TYPE "ST_SpkUnitHal"
VERSION : 0.1
   STRUCT
      CylA : "ST_SpkCylHal";
      CylB : "ST_SpkCylHal";
   END_STRUCT;

END_TYPE
